# EPICS autosave request: iocBoot/gmca_23o_ioc1/dbSave/bluiceConfig.req
$(P)waitForFeedback
$(P)enableBeamstopCheck
$(P)enableEnergyGapCheck
$(P)enableEndShutterCheck
